Fanuc KAREL source: kb00179.KL

PROGRAM KB00179
%NOLOCKGROUP
%ENVIRONMENT REGOPE
VAR
P1:INTEGER;P2 : STRING[80];P3:INTEGER
BEGIN
--
--
P1=1
P2='A'
P3=1
SET_SREG_CMT(P1,P2,P3)
END KB00179
